FUNCTION_BLOCK CL_AxisMC EXTENDS CL_CGSSystemBase
VAR
  bInit                 : BOOL := FALSE;
  _AxisDriver_R         : REFERENCE TO CL_AxisDriverAX8206;
  _stMotorAxis_R			  : REFERENCE TO AXIS_REF;//axis reference linked to I/O
  _stMasterAxis_R       : REFERENCE TO AXIS_REF;//master axis
  _stMC                 
: ST_AxisMC;
  
  _stAxisJog_R          : REFERENCE TO AXIS_REF;
  
  //private properties 
  _nStep                : E_StepMC;
  _nStepMain            : E_RequAxle := E_RequAxle.Idle;
  
  _nRequAxle            : E_RequAxle;
  _nPreviousRequ        : E_RequAxle;
  _nActualRequ          : E_RequAxle;  
  
  _bIsDone			        : BOOL := FALSE;	
  _bIsBusy			        : BOOL := FALSE;	
  _bIsPowered			      : BOOL := FALSE;
	_bError			          : BOOL := FALSE;
  _bIsAxisMaster			  : BOOL := FALSE;
	_nErrorId		          : UDINT := 0;
 
  //remove the following after debug
  _bMCBusy			        : BOOL;
  _bMCError			        : BOOL;
  _bMCStatus            : BOOL;
	//_MCerrId			        : UDINT;

  _bPowerOn             : BOOL := FALSE;
  _bGearOut             : BOOL := FALSE;
  _bStop                : BOOL := FALSE;
  _bGearInDyn           : BOOL := FALSE;
  _bJogFW               : BOOL := FALSE;
  _bJogBW               : BOOL := FALSE;
  _bIsCoupled           : BOOL := FALSE;
  
  _bExecPreviousRequ    : BOOL := FALSE;
    
	_bEnableMove          : BOOL := TRUE;   // Enable the moving of axis
	_lrAxisOverride	      : LREAL:= 100.0;  // Override of the axis velocity
  
  //_bExecJog             : BOOL := FALSE;
  //_bExecJogFWIn         : BOOL := FALSE;
  // _bExecJogBWIn         : BOOL := FALSE;
  _bJogCmdAborted       : BOOL := FALSE;
  _bAxisMovedbyJog      : BOOL := FALSE;

  _lrJogVelocity        : LREAL;
  
  _bGearInCmdAborted    : BOOL := FALSE;
  _lrMotorGearRatio     : LREAL;
  _lrAcceleration       : LREAL;
  _lrInverse            : LREAL; //Line1-Left -> _lrInverse:=1.0 while Line2-Right -> _lrInverse:=-1.0
  
  stStopProfile         : ST_AXIS_MOVE_PROFILE; //.Dec If the value is 0, the deceleration from the move command is used   .Jerk If the value is 0, the deceleration from the move command is used
 
  //counters
  _uiRetryPowerOnCnt_C  : UINT := C.uiRetryPowerOnCnt_C;  //PowerOn retry
  _uiRetryPowerOnCnt    : UINT := _uiRetryPowerOnCnt_C;  //_uiRetryPowerOnCnt_C PowerOn retry
   
  //timeout MC request
  _bRequTimeout         : BOOL;
  WaitNextState         : CL_WaitTimer; 
  
  _nJogMode             : E_JogMode;
  
  //Error handling
  //_bErrMsgShow        : BOOL := true;
  _sWhichAxis           : STRING(16);
  _nAxisErrType         : E_AxisErrorType;
END_VAR

IF bInit THEN
   This^.RunMC();//run M.otion C.ontrol (MC) FB function on entry
   THIS^.Run();
   This^.RunMC();//run M.otion C.ontrol (MC) FB function on exit, to speed-up 1 PLC cycle the refresh of the MC command
END_IF

METHOD PROTECTED InitDefect : BOOL
VAR_INPUT
END_VAR
InitDefect := true;
END_METHOD

METHOD PUBLIC InitMC : BOOL
VAR_INPUT
  stIrrLine       : ST_LineReference;
  stAxisMotor_P	  : POINTER TO AXIS_REF;
  stAxisMaster_P  : POINTER TO AXIS_REF;
  AxisDriver_P    : POINTER TO CL_AxisDriverAX8206;
END_VAR
InitMC := FALSE;
//do not check AxisDriver_P, because master axis ha no driver associated
IF stAxisMotor_P <> 0 AND stAxisMaster_P <> 0 AND NOT bInit THEN
  _bIsAxisMaster := stAxisMotor_P = stAxisMaster_P;
  
  _stMotorAxis_R REF= stAxisMotor_P^;
  _stMasterAxis_R REF= stAxisMaster_P^;
  _stAxisJog_R REF= _stMotorAxis_R;
  
  IF _bIsAxisMaster THEN
    bInit := AxisDriver_P = 0; 
    //do not assign _AxisDriver_R, because master axis has no driver associated !
  ELSE
    bInit := TRUE;
    _AxisDriver_R REF= AxisDriver_P^;
	END_IF
  
  bInit := binit AND SUPER^.InitSystemBase( IrrLine := stIrrLine, stSystemStatus_ARR := G.stSystemStatus_ARR);
  bInit := bInit AND InitParams();
  bInit := bInit AND InitDefect();
  InitMC := bInit;
END_IF
END_METHOD

METHOD PROTECTED InitParams : BOOL
VAR_INPUT
END_VAR
InitParams := true;
//if the listed parameters are equal 0.0 -> the standard parameter from the axis configuration in the System Manager is used
_lrJogVelocity := 0.3;//m/s
_nJogMode := MC_JOGMODE_STANDARD_SLOW;//MC_JOGMODE_STANDARD_FAST;  MC_JOGMODE_CONTINUOUS
_nJogMode := MC_JOGMODE_STANDARD_FAST; 
_stMC.fbMoveJog(Axis := _stMotorAxis_R, Position := 0.0, Velocity := _lrJogVelocity, Acceleration := 0.0, Deceleration := 0.0, Jerk := 0.0);
_lrInverse := 1.0;
END_METHOD

PROPERTY IsBusy : bool
GET
IsBusy := _bIsBusy;
END_GET
END_PROPERTY

PROPERTY IsDone : bool
GET
IsDone := _bIsDone;
END_GET
END_PROPERTY

PROPERTY IsDoneNoError : bool
GET
IsDoneNoError := _bIsDone and not _bError;
END_GET
END_PROPERTY

PROPERTY PUBLIC IsError : Bool
GET
IsError := _bError;
END_GET
END_PROPERTY

METHOD PUBLIC JogExec : BOOL
VAR_INPUT
  //bExecIn : BOOL := FALSE;
  bExecJogFWIn : BOOL := FALSE;
  bExecJogBWIn : BOOL := FALSE;
END_VAR
//_bExecJog := bExecIn; 
//bExecJogFWIn and bExecJogBWIn cannot be both true but they can be both false
if bExecJogFWIn <> bExecJogBWIn then
  //_bExecJogFWIn := bExecJogFWIn;
  //_bExecJogBWIn := bExecJogBWIn;
  _bJogFW := bExecJogFWIn;
  _bJogBW := bExecJogBWIn;
else
  //_bExecJogFWIn := _bExecJogBWIn := FALSE;
  _bJogFW := _bJogBW := FALSE;
END_IF
 _bAxisMovedbyJog := _stMC.fbMoveJog.Active;
 _bJogCmdAborted := _stMC.fbMoveJog.CommandAborted;
//_bJogFW := _bExecJogFWIn;
//_bJogBW := _bExecJogBWIn;
END_METHOD

PROPERTY PUBLIC nErrorID : UDINT
GET
nErrorID := _nErrorID;
END_GET
END_PROPERTY

METHOD PRIVATE OnEntryRequ
VAR_INPUT
END_VAR
_nStep := E_StepMC.Init;

_bIsBusy := TRUE;
_bIsDone := false;
_bError := FALSE;
_nErrorId	:= 0;

_bRequTimeout := false;
_bGearInCmdAborted := FALSE;
_bJogCmdAborted := false;
_bJogFW := _bJogBW := false;
_bAxisMovedbyJog := false;
//_bExecJogFWIn := _bExecJogBWIn := false;
//_bExecJog := false;
END_METHOD

METHOD PRIVATE OnExitRequError
VAR_INPUT
  ErrorIDIn     : UDINT;
  nAxisErrIn    : E_AxisErrorType;
END_VAR
_nStepMain := E_RequAxle.Error;
_bIsDone	:= TRUE;
_bIsBusy	:= FALSE;
_bError := true;
_nErrorId := ErrorIDIn;
_bExecPreviousRequ := FALSE;
_bIsPowered := FALSE;
_nAxisErrType := nAxisErrIn;
END_METHOD

METHOD PRIVATE OnExitRequOk
VAR_INPUT
END_VAR
_nStepMain := E_RequAxle.Idle;
_bIsDone	:= TRUE;
_bIsBusy	:= FALSE;
_bError := false;
_nErrorId	:= 0;
//_nRequAxle := E_RequAxle.NoRequ;//not necessary set inside method Run
END_METHOD

METHOD PRIVATE OnExitRequRetry
VAR_INPUT
  ErrorIDIn : UDINT;
  RequRetryIn  : E_RequAxle;
END_VAR
_nStepMain := E_RequAxle.Idle;
_bIsDone	:= FALSE;
_bIsBusy	:= TRUE;
_bError := true;
_nErrorId := ErrorIDIn;
_nRequAxle := RequRetryIn;
_bExecPreviousRequ := TRUE;
_bIsPowered := false;
END_METHOD

{attribute 'TcRpcEnable'}
METHOD RequGearInDyn : bool
RequGearInDyn := bInit AND _bIsPowered AND NOT _bError AND NOT _bIsBusy AND NOT _bIsAxisMaster;
//_stMotorAxis_R <> _stMasterAxis_R GearInDyn only on real axis not master axis
//_stMotorAxis_R = _stMasterAxis_R GearInDyn on virtual axis in this case make no sense
IF RequGearInDyn THEN
	_nRequAxle := E_RequAxle.GearInDyn;
else
  _nRequAxle := E_RequAxle.NoRequ;
END_IF
END_METHOD

{attribute 'TcRpcEnable'}
METHOD RequGearOut : bool
RequGearOut := bInit AND NOT _bError AND NOT _bIsBusy AND NOT _bIsAxisMaster;
//to not check _bIsPowered because the GearOut cab be executed even if not power-on
//_stMotorAxis_R <> _stMasterAxis_R GearInDyn only on real axis not master axis
//_stMotorAxis_R = _stMasterAxis_R GearInDyn on virtual axis in this case make no sense

IF RequGearOut and _bIsCoupled THEN
	_nRequAxle := E_RequAxle.GearOut;
  //request GearOut only if the axis is coupled
else
  //RequGearOut can be only false, _bIsCoupled can be true or false
  _bIsDone := not _bIsCoupled;
  //the axis was already Decoupled; only in this case set _bIsDone as the request to decouple is "virtually" executed
  //otherwise set it to false
  _nRequAxle := E_RequAxle.NoRequ;
END_IF
END_METHOD

{attribute 'TcRpcEnable'}
METHOD RequJogAxisMaster : bool
RequJogAxisMaster := bInit AND _bIsPowered AND NOT _bError AND NOT _bIsBusy AND _bIsAxisMaster;
IF RequJogAxisMaster THEN
  _stAxisJog_R := _stMasterAxis_R;//change the pointer to the Jog axis ref in order to use the master axis
	_nRequAxle := E_RequAxle.Jog;
else
  _nRequAxle := E_RequAxle.NoRequ;
END_IF
END_METHOD

{attribute 'TcRpcEnable'}
METHOD RequJogAxisMotor : bool
RequJogAxisMotor := bInit and _bIsPowered AND NOT _bError and not _bIsBusy AND NOT _bIsAxisMaster;
IF RequJogAxisMotor THEN
  _stAxisJog_R := _stMotorAxis_R;//change the pointer to the Jog axis ref in order to use the motor axis
	_nRequAxle := E_RequAxle.Jog;
else
  _nRequAxle := E_RequAxle.NoRequ;
END_IF
END_METHOD

{attribute 'TcRpcEnable'}
METHOD RequPowerOFF : BOOL
RequPowerOFF := bInit and _bIsPowered AND NOT _bError and not _bIsBusy;
IF RequPowerOFF THEN
	_nRequAxle := E_RequAxle.PowerOff;
else
  _nRequAxle := E_RequAxle.NoRequ;
END_IF
END_METHOD

{attribute 'TcRpcEnable'}
METHOD RequPowerON : bool
RequPowerON := bInit and NOT _bIsPowered AND NOT _bError and not _bIsBusy;
IF RequPowerON THEN
	_nRequAxle := E_RequAxle.PowerOn;
else
  _nRequAxle := E_RequAxle.NoRequ;
END_IF
END_METHOD

{attribute 'TcRpcEnable'}
METHOD public RequReset : bool
RequReset := bInit;//no conditions: this request is always executed -> removed bInit and NOT _bError and not _bIsBusy
IF bInit THEN
	_nRequAxle	:= E_RequAxle.Reset;
END_IF
END_METHOD

METHOD PRIVATE RequResetAndPrevious : BOOL
RequResetAndPrevious := bInit;//no conditions: this request is always executed -> removed bInit and NOT _bError and not _bIsBusy
IF bInit THEN
	_nRequAxle	:= E_RequAxle.Reset;
  _bExecPreviousRequ := TRUE;
END_IF
END_METHOD

{attribute 'TcRpcEnable'}
METHOD RequStop : bool
RequStop := bInit and _bIsPowered AND NOT _bError and not _bIsBusy;
IF RequStop THEN
	_nRequAxle := E_RequAxle.Stop;
else
  _nRequAxle := E_RequAxle.NoRequ;
END_IF
END_METHOD

METHOD PRIVATE Run
WaitNextState();
CASE _nStepMain OF
  E_RequAxle.Idle:
    IF _nRequAxle <> E_RequAxle.NoRequ THEN
      IF NOT _bExecPreviousRequ THEN
        _nPreviousRequ := _nRequAxle;
      END_IF
      _nStepMain := _nRequAxle;
      _nActualRequ := _nRequAxle;
      _nRequAxle := E_RequAxle.NoRequ;
      OnEntryRequ();
    end_if
  E_RequAxle.PowerOn : StmPowerOn_Off(bPowerOnIn := TRUE);
  E_RequAxle.PowerOff : StmPowerOn_Off(bPowerOnIn := FALSE);
  E_RequAxle.Jog : StmJog();
  E_RequAxle.GearInDyn : StmGearInDyn();
  E_RequAxle.GearOut : StmGearOut();
  E_RequAxle.Reset : StmReset();
  E_RequAxle.Error : StmError();
  E_RequAxle.Stop : StmStop();
  else;     
END_CASE
Case01Hysto(_nStepMain);
END_METHOD

METHOD PRIVATE RunMC
_stMC.fbPower(
    Axis:= _stMotorAxis_R, 
    Enable:= _bPowerOn, 
    Enable_Positive:= _bPowerOn, 
    Enable_Negative:= _bPowerOn, 
    Override:= _lrAxisOverride, 
    Status=>_bMCStatus ,
    Busy=>_bMCBusy , 
    Error=>_bMCError);
        
_stMC.fbReset(
    Axis:= _stMotorAxis_R, 
    Busy=>_bMCBusy , 
    Error=>_bMCError);

_stMC.fbMoveJog(
    Axis := _stAxisJog_R,
    JogForward := _bJogFW,
    JogBackwards := _bJogBW,
    Mode := _nJogMode,
    Velocity := _lrJogVelocity);
      
_stMC.fbGearInDyn(
    Master := _stMasterAxis_R,
    Slave:= _stMotorAxis_R,
    Enable := _bGearInDyn,//continous signal true
    GearRatio := _lrMotorGearRatio,
    Acceleration := _lrAcceleration,
    Busy=>_bMCBusy,
    Error=>_bMCError);
//ATTENTION MC_GearInDyn has Busy = Active = true until is active!

_stMC.fbGearOut(
    Slave:= _stMotorAxis_R,
    Execute := _bGearOut);//rising edge

_stMC.fbStop(
    Axis:= _stMotorAxis_R,
    Execute := _bStop);//rising edge

_bIsCoupled := _stMotorAxis_R.Status.Coupled;
   
///////////////////////////////////////////////OLD
	(*
  fbReadStatus              : MC_ReadStatus;
	fbReadAxisError				    : MC_ReadAxisError;//Status and parameter - Read Axis Error
	fbReadActualPosition			: MC_ReadActualPosition;//Status and parameter - Read Actual Position
	fbReadActualVelocity			: MC_ReadActualVelocity;//Status and parameter - Read Actual Velocity
  
 	fbSetPosition					    : MC_SetPosition;//Axis function - Set Position
	fbHome							      : MC_Home;//Home
	fbMoveAbsolute1				    : MC_MoveAbsolute;//	MC_MoveAbsolute1
  fbMoveAbsoluteWheelCheck  : MC_MoveAbsolute;// Add CustomAutomation 07.03.2023: Check du diamètre des roues 
  fbMoveAbsoluteCorrection  : MC_MoveAbsolute;// Add CustomAutomation 07.03.2023: Correction fin de parcours
 	fbMoveRelative					  : MC_MoveRelative;//Move Relative
	fbMoveVelocity					  : MC_MoveVelocity;//Move Velocity
	fbPosCorrectionLimiter    : MC_PositionCorrectionLimiter;//Special extensions - Position Correction Limiter
*)
 
(*
_stMC.fbHome(Axis:=MotorAxle^, bCalibrationCam:=_udCalibrationSensor_P^.19,
		    Options := stHomingOption, Position := lrnOffsetExtractorHoming);    
fbMoveAbso(Axis:= _AxisREF_P^);
fbReadStatus(Axis:= _AxisREF_P^,Enable := TRUE);	// Ok, actually done in the first lines.
fbMoveJog(Axis := _AxisREF_P^,JogForward := stJogControl.bMoveFW, JogBackwards := stJogControl.bMoveBW);

fbTimeRetryHomming(IN := nStep = E_StepAxis.AbortHoming);
fbTimeAbortHoming(IN := nStep = E_StepAxis.RetryHoming);
fbTrigErrorMotor(CLK := _AxisREF_P^.NcToPlc.ErrorCode <> 0);
*)
END_METHOD

METHOD PRIVATE StmError
var
  nActLine      : UINT;
  fbFormatStr	  : FB_FormatString;
  sTmp          : T_MaxString;
  sOutMsg       : T_MaxString;
  //bTmp1Err      : BOOL;
  //nErrIdOut     : UDINT;
END_VAR
_nStepMain := E_RequAxle.Idle;
//_stMC.fbPower.Enable := FALSE;
//_stMC.fbPower.Enable_Positive	:= FALSE;
//_stMC.fbPower.Enable_Negative	:= FALSE;
//fbHome.Execute := FALSE;
//fbHomeInv.Execute	:= FALSE;

if MRIrrLine <> MRIrrLineFixedID then 
  nActLine := MRIrrLineFixedID;//the real line if an HMI for each ronot is contained in MRIrrLineFixedID
else
  nActLine := MRIrrLine;
END_IF

sTmp := _sWhichAxis;  
fbFormatStr(
  sFormat	:= 'Irrigation line: %d  Axis motor: %s  MC error ID: %d  Request: ', 
  arg1  := F_UINT(nActLine),
  arg2  := F_STRING(sTmp),
  arg3	:= F_UDINT(_nErrorId),
  //bError => bTmp1Err,  
  //nErrId => nErrIdOut, 
  sOut	=> sOutMsg);

sTmp := '';
case _nActualRequ of
  E_RequAxle.PowerOn : sTmp := 'Power ON';
  E_RequAxle.PowerOff : sTmp := 'Power OFF';
  E_RequAxle.Reset : sTmp := 'Reset';
  E_RequAxle.Jog : sTmp := 'Jog';
  E_RequAxle.GearInDyn : sTmp := 'GearInDyn';
  E_RequAxle.GearOut : sTmp := 'GearOut';
  E_RequAxle.Stop : sTmp := 'Stop';
  else
    sTmp := 'Not listed';
end_case
sOutMsg := concat(sOutMsg,sTmp);

sTmp := '';
CASE _nAxisErrType OF
  E_AxisErrorType.NoError : sTmp :=' failed no error reported';
  E_AxisErrorType.MCError : sTmp :=' failed due to MC error';
  E_AxisErrorType.Retry : sTmp :=' failed after retry';
  E_AxisErrorType.Timeout : sTmp :=' timed out';
  ELSE;
END_CASE
sOutMsg := concat(sOutMsg,sTmp);
  
ADSLOGSTR(ADSLOG_MSGTYPE_LOG, 'CL_Axis error loop  %s',sOutMsg);
//ADSLOGSTR(ADSLOG_MSGTYPE_MSGBOX, 'CL_Axis error loop  %s',sOutMsg);
END_METHOD

METHOD PRIVATE StmGearInDyn
CASE _nStep OF 
  E_StepMC.Init :
    _bGearInDyn	:= TRUE;//until enable = true -> As long as "Enable" is TRUE, the gear factor can be changed cyclically
    _bGearOut := false;
    _lrMotorGearRatio := 1.0 * _lrInverse;
    _lrAcceleration := 0.0;// If the value is 0, the standard acceleration from the axis configuration in the System Manager is used
    WaitNextState.Start(C.tTimeOutAxisMC_C);
    _nStep := E_StepMC.Busy;
  
  E_StepMC.Busy :
    IF _stMC.fbGearInDyn.CommandAborted THEN
      _nStep := E_StepMC.CmdAborted;
    END_IF
    IF WaitNextState.End THEN
      _nStep := E_StepMC.Timeout;
    ELSIF _stMC.fbGearInDyn.Busy THEN //Active == Busy
      //ATTENTION MC_GearInDyn has Busy = Active = true until is active!
      _nStep := E_StepMC.End;
    END_IF
    
  E_StepMC.End:
    IF NOT _stMC.fbGearInDyn.Error THEN  
      OnExitRequOk();
    ELSE
      _bRequTimeout := false;
      OnExitRequError(_stMC.fbGearInDyn.ErrorID, E_AxisErrorType.MCError);
    END_IF
  
  E_StepMC.CmdAborted:
    _bGearInCmdAborted := true;
    OnExitRequOk();
    //OnExitRequError(_stMC.fbGearInDyn.ErrorID);
    
  E_StepMC.Timeout:
    _bRequTimeout := true;
    OnExitRequError(_stMC.fbGearInDyn.ErrorID, E_AxisErrorType.Timeout);   
end_case
END_METHOD

METHOD PRIVATE StmGearOut
CASE _nStep OF 
E_StepMC.Init :
  _bGearInDyn	:= false;
  _bGearOut := TRUE; //executed with a rising edge
  WaitNextState.Start(C.tTimeOutAxisMC_C);
  _nStep := E_StepMC.Busy;

E_StepMC.Busy :
  IF WaitNextState.End THEN
    _nStep := E_StepMC.Timeout;
  ELSIF NOT _stMC.fbGearOut.Busy THEN
    WaitNextState.Start(C.tTimeOutAxisMC_C);
    _nStep := E_StepMC.Done;
  END_IF

E_StepMC.Done :
  IF WaitNextState.End THEN
     _nStep := E_StepMC.Timeout;
  ELSIF _stMC.fbGearOut.Done THEN
    _nStep := E_StepMC.End;
  END_IF
  
E_StepMC.End:
  IF NOT _stMC.fbGearOut.Error THEN  
    _bGearOut := false;//executed with a rising edge
    OnExitRequOk();
  ELSE
    _bGearOut := false;//executed with a rising edge
    _bRequTimeout := false;
    OnExitRequError(_stMC.fbGearOut.ErrorID, E_AxisErrorType.MCError);
  END_IF

E_StepMC.Timeout:
    _stMC.fbGearOut.Execute := FALSE;
    _bRequTimeout := false;//executed with a rising edge
    OnExitRequError(_stMC.fbGearOut.ErrorID, E_AxisErrorType.Timeout);  
end_case
END_METHOD

METHOD PRIVATE StmJog
CASE _nStep OF 
  E_StepMC.Init://step by default set by OnEntryRequ method
    _bJogFW := false;//_bExecJogFWIn;
    _bJogBW := false;//_bExecJogBWIn;
    _nStep := E_StepMC.Busy;
   
  E_StepMC.Busy :    
    IF _stMC.fbMoveJog.CommandAborted THEN
      _nStep := E_StepMC.CmdAborted;
    ELSIF NOT _stMC.fbMoveJog.Busy THEN
      _nStep := E_StepMC.End;
    END_IF     
        
  E_StepMC.CmdAborted:
    _bAxisMovedbyJog := false;
    _bJogCmdAborted := true;
    //_bExecJog := false; 
    OnExitRequOk();
                          
  E_StepMC.End:
    _bJogFW := FALSE;
    _bJogBW := FALSE;
    _bAxisMovedbyJog := FALSE;
    _bJogCmdAborted := false;
    //_bExecJog := false; 
    IF NOT _stMC.fbMoveJog.Error THEN  
      OnExitRequOk();
    ELSE
      OnExitRequError(_stMC.fbMoveJog.ErrorID, E_AxisErrorType.MCError);
    end_if                  
end_case
Case02Hysto(_nStep);
END_METHOD

METHOD PRIVATE StmPowerOn_Off
VAR_INPUT
  bPowerOnIn : BOOL;
END_VAR
VAR
  b : BOOL;
END_VAR
CASE _nStep OF   
  E_StepMC.Init:
    _bPowerOn := bPowerOnIn;
    _nStep := E_StepMC.PowerOnCheckStatusError;
  
  E_StepMC.PowerOnCheckStatusError:
    b := _stMotorAxis_R.Status.Error;
    //b := TRUE;
    IF NOT b THEN //really at the level of NC Status Error flag
     _nStep := E_StepMC.Busy;
     IF _bIsAxisMaster THEN 
       WaitNextState.Start(C.tTimeOutAxisMasterMC_C);
     ELSE
       WaitNextState.Start(C.tTimeOutAxisMC_C);
		 END_IF    
     //_uiRetryPowerOnCnt := _uiRetryPowerOnCnt_C; 
    ELSE
      _nStep := E_StepMC.PowerOnRetryError;
 		END_IF
  
  E_StepMC.Busy:
    IF _stMC.fbPower.Busy THEN
      _nStep := E_StepMC.PowerOnCheckStatus;
		END_IF
    
  E_StepMC.PowerOnCheckStatus:
    b := _stMC.fbPower.Status;
    {IF defined (MiniRobotSim)}
    b := TRUE;
    {END_IF}
    IF b THEN
      b := _stMC.fbPower.Error;
      IF b THEN 
        _nStep := E_StepMC.PowerOnRetryError;
      ELSE       
        _bIsPowered := bPowerOnIn;
        OnExitRequOk();
        _uiRetryPowerOnCnt := _uiRetryPowerOnCnt_C;
        _bExecPreviousRequ := FALSE;
      END_IF
    ELSE 
      IF WaitNextState.End THEN    
        _nStep := E_StepMC.PowerOnRetryError;
      END_IF
    END_IF

  E_StepMC.PowerOnRetryError:
    //_bPowerOn := FALSE;
    IF _uiRetryPowerOnCnt = 0 THEN
      OnExitRequError(_stMC.fbPower.ErrorID, E_AxisErrorType.Retry);//after _uiRetryPowerOnCnt still impossible to PowerOn
      _uiRetryPowerOnCnt := _uiRetryPowerOnCnt_C;
      _bExecPreviousRequ := FALSE;
     ELSE
      OnExitRequRetry(ErrorIDIn := _stMC.fbPower.ErrorID, RequRetryIn := E_RequAxle.Reset);
      _uiRetryPowerOnCnt := _uiRetryPowerOnCnt - 1;
    END_IF    
END_CASE
Case02Hysto(_nStep);
END_METHOD

METHOD PRIVATE StmReset


CASE _nStep OF 
E_StepMC.Init :
  _stMC.fbReset.Execute	:= TRUE;
  WaitNextState.Start(C.tTimeOutAxisMC_C);
  _nStep := E_StepMC.Busy;

E_StepMC.Busy :
  IF WaitNextState.End THEN
    _nStep := E_StepMC.Timeout;
  ELSIF _stMC.fbReset.Busy THEN
    WaitNextState.Start(C.tTimeOutAxisMC_C);
    _nStep := E_StepMC.Done;
  END_IF

E_StepMC.Done :
  IF WaitNextState.End THEN
     _nStep := E_StepMC.Timeout;
  ELSIF _stMC.fbReset.Done THEN
    _nStep := E_StepMC.End;
  END_IF
  
E_StepMC.End:
  IF NOT _stMC.fbReset.Error THEN  
    _stMC.fbReset.Execute := FALSE;
    IF _bExecPreviousRequ THEN
      _nRequAxle := _nPreviousRequ;
      _nStepMain := E_RequAxle.Idle;
    ELSE
      OnExitRequOk();
    END_IF
  ELSE
    _stMC.fbReset.Execute := FALSE;
    _bRequTimeout := false;
    OnExitRequError(_stMC.fbReset.ErrorID, E_AxisErrorType.MCError);
  END_IF

E_StepMC.Timeout:
    _stMC.fbReset.Execute := FALSE;
    _bRequTimeout := true;
    OnExitRequError(_stMC.fbReset.ErrorID, E_AxisErrorType.Timeout);  
end_case
Case03Hysto(_nStep);
END_METHOD

METHOD PRIVATE StmStop
CASE _nStep OF 
  E_StepMC.Init:
    _bGearInDyn	:= false;
    _stMC.fbStop.Deceleration	:= stStopProfile.Dec;
    _stMC.fbStop.Jerk	:= stStopProfile.Jerk;
    _bStop := true; //executed with a rising edge
    WaitNextState.Start(C.tTimeOutAxisMC_C);
    _nStep := E_StepMC.Busy;
  
  E_StepMC.Busy:
    IF WaitNextState.End THEN
      _nStep := E_StepMC.Timeout;
    ELSIF _stMC.fbStop.Busy THEN
      WaitNextState.Start(C.tTimeOutAxisMC_C);//this timing is function of the dynamic of the whole robot!
      _nStep := E_StepMC.Stopping;
    END_IF
  
  E_StepMC.Stopping:
     IF WaitNextState.End THEN
      _nStep := E_StepMC.Timeout;
     ELSIF _stMotorAxis_R.Status.NotMoving THEN
       WaitNextState.Start(C.tTimeOutAxisMC_C);
      _nStep := E_StepMC.Stopping;
		 END_IF
     
  E_StepMC.Done:
    IF WaitNextState.End THEN
       _nStep := E_StepMC.Timeout;
    ELSIF _stMC.fbStop.Done THEN
      _nStep := E_StepMC.End;
    END_IF  
    
  E_StepMC.End:
    IF NOT _stMC.fbStop.Error THEN  
      _bStop := false;//executed with a rising edge
      OnExitRequOk();
    ELSE
      _bStop := false;//executed with a rising edge
      _bRequTimeout := false;
      OnExitRequError(_stMC.fbGearOut.ErrorID, E_AxisErrorType.MCError);
    END_IF
  
  E_StepMC.Timeout:
      _bStop := FALSE;
      _bRequTimeout := false;//executed with a rising edge
      OnExitRequError(_stMC.fbGearOut.ErrorID, E_AxisErrorType.Timeout);  
end_case
END_METHOD

END_FUNCTION_BLOCK

(* stored: Version 1.1.0.1, ProductVersion 3.1.4024.12
   POU CL_AxisMC: Id {86271131-74c3-440e-8c21-b97ff935d7af}, SpecialFunc None
   Method InitDefect: Id {69a74c5b-a8c1-48ec-ad03-8339b041f124}
   Method InitMC: Id {2947aad6-89af-4507-aa27-ffb6102c3e52}
   Method InitParams: Id {c822e9fa-eea8-4311-a8be-35f66d9b703d}
   Property IsBusy: Id {d7c98a25-7356-4fb0-9e7a-bc4c705a71dc}
   Get Get: Id {3519b6e6-03c4-40c0-b8b6-e3c5bb068ea2}
   Property IsDone: Id {96e61b31-d3fa-4cf1-8dd7-92126c3c6bef}
   Get Get: Id {8696b162-3a47-4260-a328-d7d66fd33898}
   Property IsDoneNoError: Id {510816a2-92f4-4604-af12-952b2c4f733d}
   Get Get: Id {c0a8db65-a116-4f65-9876-e8505e01d9fb}
   Property IsError: Id {34627583-c30e-46ca-ba92-abc88abb3bd8}
   Get Get: Id {df66aa41-4533-4511-bda2-aaba69b95d48}
   Method JogExec: Id {8592c973-c006-444d-93c6-86f4e3952831}
   Property nErrorID: Id {8d3317ee-d2ef-482d-a9d2-1120de114392}
   Get Get: Id {4c8c98c1-57ac-4c73-be1f-aad427892288}
   Method OnEntryRequ: Id {230d5f2c-93b6-4eb8-bd24-5b6b55e6476e}
   Method OnExitRequError: Id {d015decd-a857-4c36-a77e-6afbb638a30b}
   Method OnExitRequOk: Id {a0389a39-6280-4762-8dbf-2b24b6c17de9}
   Method OnExitRequRetry: Id {35ef2c45-9e1b-41f8-89f3-49d969d38279}
   Method RequGearInDyn: Id {903517ee-9ade-42de-abc9-5c6fcd098db3}
   Method RequGearOut: Id {60abab3f-91df-4b45-93f2-9e732c64f765}
   Method RequJogAxisMaster: Id {7c24f518-fbdc-4e8f-95c9-e66859ad42bc}
   Method RequJogAxisMotor: Id {85c2f71d-4215-4e1e-b9e2-dae88d863f58}
   Method RequPowerOFF: Id {d948d7ed-314b-49f1-b56a-12ed03f0cdb3}
   Method RequPowerON: Id {dc2d922e-ed56-44a2-b5f2-59d0d0a6f03d}
   Method RequReset: Id {abbde50c-809d-4a9a-81e4-a38006b3b251}
   Method RequResetAndPrevious: Id {806b90d6-d512-4e95-9992-33d3c953fe31}
   Method RequStop: Id {0e701679-6dcc-400c-a87c-3ea674ae4664}
   Method Run: Id {5ea0ba84-4411-4ae2-b784-f4b1dd20fb56}
   Method RunMC: Id {effdf679-c8e9-4b8a-be02-83c601485a94}
   Method StmError: Id {87aea61f-b034-476e-8424-5557144e0f3e}
   Method StmGearInDyn: Id {9a3ea223-c254-4297-9010-6a65a69a26e6}
   Method StmGearOut: Id {7fc9b694-1dc7-49ad-acb4-c03aed63ee35}
   Method StmJog: Id {328921f4-fe55-4ae8-8f95-7c67258651dc}
   Method StmPowerOn_Off: Id {af9b62a9-996e-4f71-ad22-22899f2dc5e1}
   Method StmReset: Id {752c42b5-45d9-41b7-a20c-71af002eb088}
   Method StmStop: Id {907e788a-6c6a-4519-bbdd-4a9c8e098fa5} *)
